// Mitsubishi GX Works2 project: 21   PLC: FX3G

// task Task_01 (event TRUE, interval 0, priority 31): POU_01

PROGRAM POU_01
VAR
  rt1 : R_TRIG;
  rt2 : R_TRIG;
  rt3 : R_TRIG;
  wstep : INT;
  counter : INT;
  ton1 : TON;
END_VAR
M99 := FALSE AND
M0 AND M1 AND M2 AND
Y0 AND Y1 AND Y2 AND Y3;

IF M8002 THEN
	wstep := 0;
END_IF;

rt1(_clk := M0);
rt2(_clk := M1);
rt3(_clk := M2);

IF rt1.q THEN
	ton1(in := FALSE);
	counter := 0;
	wstep := 1;
END_IF;

IF rt2.q THEN
	ton1(in := FALSE);
	counter := 0;
	wstep := 2;
END_IF;

IF rt3.q THEN
	ton1(in := FALSE);
	counter := 0;
	wstep := 3;
END_IF;

CASE wstep OF
	1:
		ton1(in := NOT ton1.q, pt := t#0.5s);
		IF ton1.q THEN
			counter := counter + 1;
			counter := counter MOD 4;
		END_IF;		
		
		zrst(TRUE, Y0, Y3);
		Z0 := counter;
		Y0Z0 := TRUE;
		
	2:
		ton1(in := NOT ton1.q, pt := t#1s);
		IF ton1.q THEN
			counter := counter + 1;
			counter := counter MOD 4;
		END_IF;		
		
		zrst(TRUE, Y0, Y3);
		Z0 := counter;
		Y0Z0 := TRUE;
	
	3:
		ton1(in := NOT ton1.q, pt := t#1.5s);
		IF ton1.q THEN
			counter := counter + 1;
			counter := counter MOD 4;
		END_IF;		
		
		zrst(TRUE, Y0, Y3);
		Z0 := counter;
		Y0Z0 := TRUE;
END_CASE;
END_PROGRAM
